FUNCTION_BLOCK FB_TcMatSimObject_1
VAR_INPUT
	/// set this flag to write FB input values to the TcComObject's input DataAreas. This will overwrite the mapped input values before module execution. Set to FALSE to read the mapped input values from the TcComObject to the FB.
	bWriteFbInputValues: BOOL := TRUE;
END_VAR
VAR
	/// process image src and dst pointers and sizes
	pDataAreas: POINTER TO ST_TcMatSimObjectDataAreaInfo;
	nDataAreas: UDINT;
	/// global interface pointers
	ipObjSrv: ITComObjectServer;
	/// object interface pointers
	ipTcComObj: ITComObject;
	ipTcCyclic: ITcCyclic;
	ipTcPostCyclic: ITcPostCyclic;
	ipTcAdi: ITcADI;
	/// task interface pointers
	ipTask: ITcTask;
	/// initial parameters
	pInitData: POINTER TO TComInitDataHdr;
	/// hResult of interface calls (0 if no error)
	hResult: HRESULT;
	/// module class ID
	moduleClsId: CLSID;
	/// expected/desired module class ID
	assignedClsId: CLSID;
	bClassIdVerified: BOOL;
	/// flag indicating whether the module instance was created dynamically
	bDynInstance: BOOL;
	/// the object state at the time FB_init was called, FB_exit will try to switch to this state (only if this means to shift down)
	eInitialObjState: TCOM_STATE := TCOM_STATE.TCOM_STATE_INIT;
END_VAR

METHOD PUBLIC AssignClassId
VAR_INPUT
	clsId : CLSID;
END_VAR
assignedClsId := clsId;
bClassIdVerified := false;
END_METHOD

PROPERTY ClassId : CLSID
GET
hResult := ReadModuleClassId();
ClassId := moduleClsId;
END_GET
END_PROPERTY

PROPERTY Error : BOOL
GET
Error := FAILED(hResult);
END_GET
END_PROPERTY

PROPERTY ErrorCode : HRESULT
GET
ErrorCode := hResult;
END_GET
END_PROPERTY

{attribute 'object_name' := 'Execute'}
METHOD Execute : HRESULT
VAR
	nDaIdx: UDINT;
	pCurDataArea: POINTER TO ST_TcMatSimObjectDataAreaInfo;
END_VAR

IF (SUCCEEDED(hResult)) THEN
  hResult := VerifyClassId();
END_IF

IF (SUCCEEDED(hResult) AND State<>TCOM_STATE_OP) THEN
  hResult := Tc2_System.E_HRESULTAdsErr.NOTREADY;
END_IF

// get image pointers
IF (SUCCEEDED(hResult)) THEN
  GetImagePtrs(hResult);
END_IF

// copy inputs
IF (pDataAreas<>0 AND bWriteFbInputValues) THEN
  FOR nDaIdx:=0 TO nDataAreas-1 DO
    IF (FAILED(hResult))THEN
      CONTINUE;
    END_IF
    pCurDataArea := pDataAreas + nDaIdx*SIZEOF(ST_TcMatSimObjectDataAreaInfo);
    IF ((pCurDataArea^.eDataAreaType <> E_TcMatSimDataAreaType.InputDst))THEN
      CONTINUE;
    END_IF
    IF (pCurDataArea^.pModuleProcImg<>0 AND pCurDataArea^.pPlcVar<>0) THEN
      MEMCPY(pCurDataArea^.pModuleProcImg,pCurDataArea^.pPlcVar,pCurDataArea^.nSize);
    ELSE
      hResult := Tc2_System.E_HRESULTAdsErr.NOINTERFACE;
    END_IF
  END_FOR
END_IF

// call cycle update
IF (SUCCEEDED(hResult)) THEN
  IF (ipTcCyclic<>0) THEN
    hResult := ipTcCyclic.CycleUpdate(ipTask:= ipTask, ipCaller:= 0, context:= 0);
  ELSE
    hResult := Tc2_System.E_HRESULTAdsErr.NOINTERFACE;
  END_IF
END_IF

// copy outputs
IF (pDataAreas<>0) THEN
  FOR nDaIdx:=0 TO nDataAreas-1 DO
    IF (FAILED(hResult))THEN
      CONTINUE;
    END_IF
    pCurDataArea := pDataAreas + nDaIdx*SIZEOF(ST_TcMatSimObjectDataAreaInfo);
    IF ((pCurDataArea^.eDataAreaType = E_TcMatSimDataAreaType.OutputSrc) OR NOT bWriteFbInputValues) THEN
      IF (pCurDataArea^.pModuleProcImg<>0 AND pCurDataArea^.pPlcVar<>0) THEN
        MEMCPY(pCurDataArea^.pPlcVar,pCurDataArea^.pModuleProcImg,pCurDataArea^.nSize);
      ELSE
        hResult := Tc2_System.E_HRESULTAdsErr.NOINTERFACE;
      END_IF
    END_IF
  END_FOR
END_IF


// call post cyclic update
IF (SUCCEEDED(hResult)) THEN
  IF (ipTcPostCyclic<>0) THEN
    hResult := ipTcPostCyclic.PostCyclicUpdate(ipTask:= 0, ipCaller:= 0, context:= 0);
  ELSE
    hResult := Tc2_System.E_HRESULTAdsErr.NOINTERFACE;
  END_IF
END_IF

ReleaseImagePtrs();

Execute := hResult;
END_METHOD

{attribute 'object_name' := 'FB_exit'}
METHOD FB_exit : BOOL
VAR_INPUT
	/// Online Change
	bInCopyCode: BOOL;
END_VAR

IF (NOT bInCopyCode) THEN
  IF (ipObjSrv<>0) THEN
    ipObjSrv.TcRelease();
    ipObjSrv := 0;
  END_IF

  ReleaseTcComInterface();
END_IF
END_METHOD

{attribute 'object_name' := 'FB_init'}
METHOD FB_init : BOOL
VAR_INPUT
	/// init retain variables
	bInitRetains: BOOL;
	/// Online Change
	bInCopyCode: BOOL;
	oid: OTCID;
END_VAR

FB_init := SUCCEEDED(Init(oid));
END_METHOD

{attribute 'object_name' := 'GetImagePtrs'}
METHOD PRIVATE GetImagePtrs
VAR_INPUT
	hr: REFERENCE TO HRESULT;
END_VAR
VAR
	nDaIdx: UDINT;
	pCurDataArea: POINTER TO ST_TcMatSimObjectDataAreaInfo;
END_VAR

IF (ipTcAdi=0) THEN
  hr := Tc2_System.E_HRESULTAdsErr.NOINTERFACE;
END_IF
IF(State<>TCOM_STATE_OP)THEN
  hr := Tc2_System.E_HRESULTAdsErr.INVALIDSTATE;
END_IF


// get pointers to process images
IF (pDataAreas<>0) THEN
  FOR nDaIdx:=0 TO nDataAreas-1 DO
    pCurDataArea := pDataAreas + nDaIdx*SIZEOF(ST_TcMatSimObjectDataAreaInfo);
    IF (FAILED(hr))THEN
      CONTINUE;
    END_IF
    IF ((pCurDataArea^.eDataAreaType <> E_TcMatSimDataAreaType.InputDst) AND (pCurDataArea^.eDataAreaType <> E_TcMatSimDataAreaType.OutputSrc))THEN
      CONTINUE;
    END_IF
    IF (pCurDataArea^.pModuleProcImg=0 AND pCurDataArea^.nSize>0) THEN
      hr := ipTcAdi.GetImagePtr(size:= pCurDataArea^.nSize , offs:=0 , adi_x:=pCurDataArea^.nDataAreaId , ppData:=ADR(pCurDataArea^.pModuleProcImg));
    END_IF
  END_FOR
END_IF

IF (FAILED(hr)) THEN
  ReleaseImagePtrs();
END_IF
END_METHOD

{attribute 'object_name' := 'GetObjPara'}
METHOD GetObjPara : HRESULT
VAR_INPUT
	pid: PTCID;
	nData: UDINT;
	pData: PVOID;
END_VAR

IF (ipTcComObj=0) THEN
  GetObjPara := Tc2_System.E_HRESULTAdsErr.NOINTERFACE;
END_IF

IF (SUCCEEDED(GetObjPara)) THEN
  GetObjPara := ipTcComObj.TcGetObjPara(pid:=pid,nData,pData,0);
END_IF
END_METHOD

{attribute 'object_name' := 'Init'}
METHOD PROTECTED Init : HRESULT
VAR_INPUT
	oid: OTCID;
END_VAR

// preinitialize variables
memset(ADR(moduleClsId),0,SIZEOF(moduleClsId));
bClassIdVerified := FALSE;
hResult := Tc2_System.E_HRESULTAdsErr.HRESULT_ADS_NOERROR;

// get object server
IF (ipObjSrv=0) THEN
  hResult := FW_ObjMgr_GetObjectServer(_AppInfo.ObjId,ADR(ipObjSrv));
END_IF

// try to get object interfaces
IF (SUCCEEDED(hresult)) THEN
  QueryTcComInterface(hResult,oid);
END_IF

// verify class id
IF (SUCCEEDED(hresult)) THEN
  hresult := VerifyClassId();
END_IF

// query interfaces, if the current state is higher than INIT
IF (SUCCEEDED(hresult) AND State>TCOM_STATE.TCOM_STATE_INIT) THEN
  QueryObjInterfaces(hResult);
END_IF

// return value
Init := hresult;
END_METHOD

{attribute 'object_name' := 'InitObjName'}
METHOD PRIVATE InitObjName
VAR_INPUT
	hr: REFERENCE TO HRESULT;
END_VAR
VAR
	objectName: STRING(255) := 'TempContr_PlcRtFbInstance';
	oid: OTCID;
END_VAR

IF (SUCCEEDED(hr)) THEN
  hr := ipTcComObj.TcGetObjectId(oid);
END_IF

IF (SUCCEEDED(hr) and bDynInstance) THEN
  objectName := TC2_STANDARD.CONCAT(objectName,'_');
  objectName := TC2_STANDARD.CONCAT(objectName,UDINT_TO_STRING(oid));
  hr := ipTcComObj.TcSetObjectName(ADR(objectName));
END_IF
END_METHOD

{attribute 'object_name' := 'Internal_SetObjState'}
METHOD PROTECTED Internal_SetObjState
VAR_INPUT
	hr: REFERENCE TO HRESULT;
	nextState: TCOM_STATE;
END_VAR

// verify class id
IF (SUCCEEDED(hr)) THEN
  hr := VerifyClassId();
END_IF

// switch object state
IF (SUCCEEDED(hr) AND nextState>=TCOM_STATE_INIT) THEN
  IF (ipTcComObj=0) THEN
    hr := Tc2_System.E_HRESULTAdsErr.NOINTERFACE;
  END_IF
  IF (ipObjSrv=0) THEN
    hr := Tc2_System.E_HRESULTAdsErr.NOINTERFACE;
  END_IF
  IF (SUCCEEDED(hr)) THEN
    hr := ipTcComObj.TcSetObjState(nextState,ipObjSrv,pInitData);
  END_IF
END_IF
END_METHOD

{attribute 'object_name' := 'QueryObjInterface'}
METHOD PRIVATE QueryObjInterface
VAR_INPUT
	hr: REFERENCE TO HRESULT;
	iid: REFERENCE TO IID;
	pipItf: POINTER TO ITcUnknown;
END_VAR
VAR CONSTANT
	pNull: PVOID := 0;
END_VAR

IF (SUCCEEDED(hr)) THEN
  IF (ipTcComObj=0) THEN
    hr := Tc2_System.E_HRESULTAdsErr.NOINTERFACE;
  ELSIF (pipItf^=ULINT_TO_DWORD(pNull)) THEN
    hr := ipTcComObj.TcQueryInterface(iid:= iid, pipItf:=pipItf);
  END_IF
END_IF
END_METHOD

{attribute 'object_name' := 'QueryObjInterfaces'}
METHOD PRIVATE QueryObjInterfaces
VAR_INPUT
	hr: REFERENCE TO HRESULT;
END_VAR

IF(State<TCOM_STATE_PREOP)THEN
  hr := Tc2_System.E_HRESULTAdsErr.INVALIDSTATE;
END_IF

//cyclic interface
QueryObjInterface(hr,IID_ITCCYCLIC,ADR(ipTcCyclic));
//post cyclic interface
QueryObjInterface(hr,IID_ITCPOSTCYCLIC,ADR(ipTcPostCyclic));
//adi interface
QueryObjInterface(hr,IID_ITcADI,ADR(ipTcAdi));
END_METHOD

{attribute 'object_name' := 'QueryTcComInterface'}
METHOD PRIVATE QueryTcComInterface
VAR_INPUT
	hr: REFERENCE TO HRESULT;
	oid: OTCID;
END_VAR

IF (ipObjSrv=0) THEN
  hr := Tc2_System.E_HRESULTAdsErr.NOINTERFACE;
END_IF

IF (SUCCEEDED(hr) AND ipTcComObj=0) THEN
  bDynInstance := FALSE;
  IF(oid>0) THEN
    // query interface of existing object
    hr := ipObjSrv.TcQueryObjectInterface(oid,IID_ITComObject,ADR(ipTcComObj));
  ELSE
    // create new instance and get the object interface
    hr := ipObjSrv.TcCreateInstance(assignedClsId,IID_ITComObject,ADR(ipTcComObj));
    IF (SUCCEEDED(hr)) THEN
      bDynInstance := TRUE;
      hr := ipTcComObj.TcSetObjectId(OTCID_CreateNewId);
    END_IF
  END_IF
  IF (SUCCEEDED(hr)) THEN
    eInitialObjState := State;
  END_IF
END_IF
END_METHOD

{attribute 'object_name' := 'ReadModuleClassId'}
METHOD PRIVATE ReadModuleClassId : HRESULT
VAR
	emptyClsId: CLSID;
END_VAR
memset(ADR(emptyClsId),0,SIZEOF(emptyClsId));
IF (memcmp(ADR(moduleClsId),ADR(emptyClsId),SIZEOF(moduleClsId))=0) THEN
  IF (ipTcComObj=0) THEN
    ReadModuleClassId := Tc2_System.E_HRESULTAdsErr.NOINTERFACE;
  END_IF

  //objectClsId := clsid;
  IF (SUCCEEDED(ReadModuleClassId)) THEN
    ReadModuleClassId := ipTcComObj.GetClassId(moduleClsId);
  END_IF
END_IF
END_METHOD

{attribute 'object_name' := 'ReleaseImagePtrs'}
METHOD PRIVATE ReleaseImagePtrs : HRESULT
VAR
	nDaIdx: UDINT;
	pCurDataArea: POINTER TO ST_TcMatSimObjectDataAreaInfo;
END_VAR

IF (ipTcAdi=0) THEN
  ReleaseImagePtrs := Tc2_System.E_HRESULTAdsErr.NOINTERFACE;
END_IF

IF (SUCCEEDED(ReleaseImagePtrs) AND pDataAreas<>0) THEN
  // release pointers to the simulink module process images
  FOR nDaIdx:=0 TO nDataAreas-1 DO
    pCurDataArea := pDataAreas + nDaIdx*SIZEOF(ST_TcMatSimObjectDataAreaInfo);

    IF (pCurDataArea^.pModuleProcImg<>0) THEN
      ipTcAdi.ReleaseImagePtr(pData:=pCurDataArea^.pModuleProcImg);
      pCurDataArea^.pModuleProcImg := 0;
    END_IF
  END_FOR
END_IF
END_METHOD

{attribute 'object_name' := 'ReleaseObjInterfaces'}
METHOD PRIVATE ReleaseObjInterfaces : HRESULT

// release interface pointers
IF (ipTcCyclic<>0) THEN
  ipTcCyclic.TcRelease();
  ipTcCyclic := 0;
END_IF
IF (ipTcPostCyclic<>0) THEN
  ipTcPostCyclic.TcRelease();
  ipTcPostCyclic := 0;
END_IF
IF (ipTcAdi<>0) THEN
  ipTcAdi.TcRelease();
  ipTcAdi := 0;
END_IF
END_METHOD

{attribute 'object_name' := 'ReleaseTcComInterface'}
METHOD PRIVATE ReleaseTcComInterface : HRESULT
VAR
	nStateChangeCnt: DINT := 0;
END_VAR

IF (ipTcComObj<>0) THEN
  WHILE (State>eInitialObjState AND nStateChangeCnt<1000) DO
    State := eInitialObjState;
    nStateChangeCnt := nStateChangeCnt+1;
  END_WHILE
  ReleaseObjInterfaces();
  IF (bDynInstance) THEN
    ReleaseTcComInterface := TC3_MODULE.FW_ObjMgr_DeleteInstance(ADR(ipTcComObj));
  ELSE
    ipTcComObj.TcRelease();
  END_IF
  ipTcComObj := 0;
END_IF
END_METHOD

{attribute 'object_name' := 'ResetHresult'}
METHOD ResetHresult
hResult := S_OK;
END_METHOD

{attribute 'object_name' := 'SaveOnlineParametersForInit'}
METHOD SaveOnlineParametersForInit : HRESULT
VAR
	idx: UINT;
	pInitElemHdr: POINTER TO TComInitDataElmHdr;
	pData: PVOID;
	nData: UDINT;
END_VAR
VAR CONSTANT
	nInitDataAlignment: UDINT := 4;
END_VAR
IF (pInitData<>0) THEN
  pInitElemHdr := pInitData + SIZEOF(pInitData^);
  FOR idx:=1 TO pInitData^.uiElmCnt DO
    pData := pInitElemHdr + ULINT_TO_DWORD(SIZEOF(pInitElemHdr^));
    nData := pInitElemHdr^.cbData;
    SaveOnlineParametersForInit := GetObjPara(pInitElemHdr^.indexOffset,nData,pData);
    IF (FAILED(SaveOnlineParametersForInit)) THEN
      RETURN;
    END_IF
    pInitElemHdr := pData + (nInitDataAlignment*((nData + nInitDataAlignment - 1)/nInitDataAlignment));
  END_FOR
ELSE
	SaveOnlineParametersForInit := Tc2_System.E_HRESULTAdsErr.NOTINIT;
END_IF
END_METHOD


METHOD PUBLIC SetDataAreaInfo
VAR_INPUT
  pDataAreas: POINTER TO ST_TcMatSimObjectDataAreaInfo;
  nDataAreas: UDINT;
END_VAR

THIS^.nDataAreas := nDataAreas;
THIS^.pDataAreas := pDataAreas;
END_METHOD


METHOD PUBLIC SetInitDataInfo
VAR_INPUT
  pInitData : POINTER TO TComInitDataHdr;
END_VAR
this^.pInitData := pInitData;
END_METHOD

{attribute 'object_name' := 'SetObjPara'}
METHOD SetObjPara : HRESULT
VAR_INPUT
	pid: PTCID;
	nData: UDINT;
	pData: PVOID;
END_VAR

IF (ipTcComObj=0) THEN
  SetObjPara := Tc2_System.E_HRESULTAdsErr.NOINTERFACE;
END_IF

IF (SUCCEEDED(SetObjPara)) THEN
  SetObjPara := ipTcComObj.TcSetObjPara(pid:=pid,nData,pData,0);
END_IF
END_METHOD

{attribute 'object_name' := 'SetObjState'}
METHOD SetObjState : HRESULT
VAR_INPUT
	finalState: TCOM_STATE;
END_VAR
VAR
	bShiftUp: BOOL;
	bShiftDown: BOOL;
	currentState: TCOM_STATE;
END_VAR

currentState := State;

bShiftUp := finalState>currentState;
bShiftDown := finalState<currentState;

// do not switch up on error
IF (FAILED(hresult)) THEN
  bShiftUp := FALSE;
END_IF
// reset existing error on switching down
IF (bShiftDown) THEN
  ResetHresult();
END_IF

// prepared state switch
CASE currentState OF
  TCOM_STATE_INIT:
    IF(bShiftUp) THEN
      QueryTcComInterface(hResult,0);
      Internal_SetObjState(hResult,TCOM_STATE.TCOM_STATE_PREOP);
      InitObjName(hResult);
    END_IF

  TCOM_STATE_PREOP:
    IF(bShiftUp) THEN
      Internal_SetObjState(hResult,TCOM_STATE.TCOM_STATE_SAFEOP);
      QueryObjInterfaces(hResult);
    ELSIF (bShiftDown) THEN
      Internal_SetObjState(hResult,TCOM_STATE.TCOM_STATE_INIT);
    END_IF

  TCOM_STATE_SAFEOP:
    IF(bShiftUp) THEN
      Internal_SetObjState(hResult,TCOM_STATE.TCOM_STATE_OP);
      QueryObjInterfaces(hResult);
    ELSIF (bShiftDown) THEN
      Internal_SetObjState(hResult,TCOM_STATE.TCOM_STATE_PREOP);
      ReleaseObjInterfaces();
    END_IF


  TCOM_STATE_OP:
    IF (bShiftDown) THEN
      Internal_SetObjState(hResult,TCOM_STATE.TCOM_STATE_SAFEOP);
    END_IF
END_CASE

SetObjState := hResult;
END_METHOD

PROPERTY State : TCOM_STATE
GET
VAR
	hr: HRESULT := S_OK;
	eObjState: TCOM_STATE;
END_VAR

IF (ipTcComObj<>0) THEN
  hr := ipTcComObj.TcGetObjState(ADR(eObjState));
IF (FAILED(hr)) THEN
  eObjState := TCOM_STATE.TCOM_STATE_INIT;
END_IF
ELSE
  eObjState := TCOM_STATE.TCOM_STATE_INIT;
END_IF
State := eObjState;
END_GET
SET
SetObjState(State);
END_SET
END_PROPERTY

{attribute 'object_name' := 'VerifyClassId'}
METHOD PRIVATE VerifyClassId : HRESULT
VAR
	emptyClsId: CLSID;
END_VAR
memset(ADR(emptyClsId),0,SIZEOF(emptyClsId));
IF (bClassIdVerified) THEN
  // class ID was already verified
  VerifyClassId := Tc2_System.E_HRESULTAdsErr.HRESULT_ADS_NOERROR;
ELSIF (memcmp(ADR(assignedClsId),ADR(emptyClsId),SIZEOF(assignedClsId))=0) THEN
  // skip class ID verification if no assignedClsId specified
  VerifyClassId := Tc2_System.E_HRESULTAdsErr.HRESULT_ADS_NOERROR;
ELSE
  // verify class ID
  VerifyClassId := ReadModuleClassId();

  IF (SUCCEEDED(VerifyClassId)) THEN
    IF (memcmp(ADR(assignedClsId),ADR(moduleClsId),SIZEOF(assignedClsId))<>0) THEN
     VerifyClassId := Tc2_System.E_HRESULTAdsErr.INVALIDCLSID;
    END_IF
  END_IF
  bClassIdVerified := SUCCEEDED(VerifyClassId);
END_IF
END_METHOD

END_FUNCTION_BLOCK

(* stored: Version 1.1.0.1, ProductVersion 3.1.4020.12
   POU FB_TcMatSimObject_1: Id {ca7fe5ec-33b5-47bb-a277-2a587f75d77a}, SpecialFunc None
   Method AssignClassId: Id {28312a73-16c9-4435-a6b6-9fe6085b9d83}
   Property ClassId: Id {63d517f0-29bc-4aca-ba6b-a37012832df6}
   Get Get: Id {156f7bac-e39e-4f44-a135-3f56ce200680}
   Property Error: Id {49f89d7e-1885-457c-a6fb-ffe2f0b11b47}
   Get Get: Id {303f12f3-cc34-4038-980d-9d1bc683d2f4}
   Property ErrorCode: Id {e159b280-7b90-428b-8c8b-22ecbb655773}
   Get Get: Id {beacc864-ac50-47cb-a449-e9ae30284b50}
   Method Execute: Id {53d9189b-3438-4efe-8ef8-c335ec4dd40e}
   Method FB_exit: Id {180a7fa7-d3df-4a41-8e95-3ef32633723b}
   Method FB_init: Id {6466ba0a-3a96-49a0-9b3a-695bfa72bd76}
   Method GetImagePtrs: Id {400172bd-9186-4ce3-ba39-246bfce0d544}
   Method GetObjPara: Id {1d8bc8b0-bf9e-40c1-b795-fe1cfcf90422}
   Method Init: Id {d4585564-01fd-482c-98b1-545b45c3a9c7}
   Method InitObjName: Id {9e27509a-88f1-4d9f-bf28-3da504e58a10}
   Method Internal_SetObjState: Id {66a31289-39ec-4f25-bb7c-153e2529a7ec}
   Method QueryObjInterface: Id {8ef370d9-ee52-431b-a47b-8660353a14a3}
   Method QueryObjInterfaces: Id {49ac6ed0-8c57-46be-8690-ff2c1fe12888}
   Method QueryTcComInterface: Id {710de71e-966e-4f96-a956-aba6a61a9827}
   Method ReadModuleClassId: Id {cb9ad669-df28-4b9c-8623-53d54d966871}
   Method ReleaseImagePtrs: Id {e3ce3625-0c77-432d-96dc-a9e929618d71}
   Method ReleaseObjInterfaces: Id {ddc66bee-92e6-4c2e-93b1-5bbfbb8e3a29}
   Method ReleaseTcComInterface: Id {087d470e-9da8-4191-9e3e-a849a4f5ab27}
   Method ResetHresult: Id {ab630a39-de38-4637-8cf3-e00929b91734}
   Method SaveOnlineParametersForInit: Id {5ca583a7-f5fc-4915-84bb-abe0bbf76e41}
   Method SetDataAreaInfo: Id {ae8caa64-c313-4dea-89c0-a5bc919544c3}
   Method SetInitDataInfo: Id {3136f0d4-0ff6-47a8-916e-f7c19c522499}
   Method SetObjPara: Id {39d4dd24-6029-4faa-bcaa-e7be4456888d}
   Method SetObjState: Id {5ab48f0e-97d5-4da0-afb9-37dc7a680ec2}
   Property State: Id {8f9b115c-ea2b-4656-85b6-dfd18f0c2e35}
   Get Get: Id {40fc1cf3-1ba0-4807-8c74-dd1e35c3d10b}
   Set Set: Id {3f8e84d9-86ac-405e-9169-6401058ec57d}
   Method VerifyClassId: Id {a47a28bd-c5a2-47d4-b64b-c157105f6a32} *)
